(* CoDeSys 2.3.9.59 project: Proyecto_Maquina_Expendedora.pro *)
(* Libraries: Standard.LIB, Iecsfc.lib 2.6.14 11:37:46 *)

(* Global variable list: Global_Variables *)
VAR_GLOBAL
(*ENTRADAS*)
	boton1:BOOL;
	boton2:BOOL;
	boton3:BOOL;
	boton4:BOOL;
	boton5:BOOL;
	boton6:BOOL;
	diezcent:BOOL;
	cincucent:BOOL;
	ciencent:BOOL;
	selector1:BOOL;
	selector2:BOOL;
	selector3:BOOL;
	selector4:BOOL;
	selector5:BOOL;
	selector6:BOOL;
	M:BOOL;
	P:BOOL;
	devolucion:BOOL;
	atasca:BOOL;
	rearme:BOOL;
	auto:BOOL;
	recogeobjeto:BOOL;
	recogecambio:BOOL;
	seleccionado:INT;
	abrir:BOOL;
(*SALIDAS*)
	dispensador1:BOOL;
	dispensador2:BOOL;
	dispensador3:BOOL;
	dispensador4:BOOL;
	dispensador5:BOOL;
	dispensador6:BOOL;
	dinero:REAL;
	cambio:REAL;
	precio:REAL;
	display:REAL;
	puertacerrada: BOOL:=TRUE;
	objetoabajo: BOOL:=FALSE;
	fila1cae:BOOL;
	fila2cae:BOOL;
	fila3cae:BOOL;
	muestradinero:BOOL;
	muestracambio:BOOL;
	luzcae:BOOL;
	luzabajo:BOOL;
	resetobjeto:BOOL;
	emergencia:BOOL;
(*CONSTANTES*)
	precio1:REAL:=1.00;
	precio2:REAL:=1.30;
	precio3:REAL:=0.80;
	precio4:REAL:=1.60;
	precio5:REAL:=2.00;
	precio6:REAL:=0.90;

(*ESTADOS*)
	metedinero: BOOL;
	sacadinero: BOOL;
	caeobjeto: BOOL;
END_VAR

(* POU PLC_PRG, ST *)
PROGRAM PLC_PRG
VAR
	inicio:BOOL:=TRUE;
	camux: INT;
	camuy:INT;
	kinderx:INT;
	kindery:INT;
	chocox:INT;
	chocoy:INT;
	bullx:INT;
	bully:INT;
	mangox:INT;
	mangoy:INT;
	kitkatx:INT;
	kitkaty:INT;
	TEMPprecio: TON;
	apaga: F_TRIG;
	apagando: BOOL;
	color:DWORD;
END_VAR
(* Selector para mostrar dinero *)
IF (inicio) THEN
	precio:=0;
	inicio:=FALSE;
END_IF
apaga (CLK := (selector1 OR selector2 OR selector3 OR selector4 OR selector5 OR selector6));
IF apaga.Q THEN apagando := TRUE; END_IF
IF selector1 THEN precio := precio1; apagando := FALSE;
ELSIF selector2 THEN precio := precio2; apagando := FALSE;
ELSIF selector3 THEN precio := precio3; apagando := FALSE;
ELSIF selector4 THEN precio := precio4; apagando := FALSE;
ELSIF selector5 THEN precio := precio5; apagando := FALSE;
ELSIF selector6 THEN precio := precio6; apagando := FALSE;
END_IF

TEMPprecio(IN:= apagando, PT:=T#3s) ;
	IF TEMPprecio.Q THEN
		seleccionado := 0;
		precio := 0;
		apagando := FALSE;
	END_IF

(* Selector para mostrar dinero disponible o cambio dependiendo del estado *)
IF muestradinero THEN display := dinero;
ELSIF muestracambio THEN display := cambio;
ELSE display := 0.00;
END_IF

(* Dependiendo de cuál se elija, cae uno u otro *)
IF (auto AND NOT objetoabajo) OR NOT auto THEN
IF (dispensador1 = TRUE) AND (camuy<=545) THEN camuy := camuy + 10; fila1cae := TRUE;
	IF (camuy = 550) THEN
		objetoabajo:=TRUE;
		fila1cae:=FALSE;
	END_IF
ELSIF (dispensador2 = TRUE) AND (kindery <=545)THEN kindery := kindery + 10; fila1cae:=TRUE;
	IF (kindery = 550) THEN
		objetoabajo := TRUE;
		fila1cae:=FALSE;
	END_IF;
ELSIF (dispensador3 = TRUE) AND (chocoy<=395) THEN chocoy := chocoy + 10; fila2cae:=TRUE;
	IF (chocoy = 400) THEN
		objetoabajo:=TRUE;
		fila2cae:=FALSE;
	END_IF
ELSIF (dispensador4 = TRUE) AND (bully <= 395) THEN bully := bully + 10; fila2cae:=TRUE;
	IF (bully = 400) THEN
		objetoabajo:=TRUE;
		fila2cae:=FALSE;
	END_IF
ELSIF (dispensador5 = TRUE) AND (mangoy <= 255) THEN mangoy := mangoy + 10; fila3cae:=TRUE;
	IF (mangoy = 260) THEN
		objetoabajo:=TRUE;
		fila3cae:=FALSE;
	END_IF
ELSIF (dispensador6 = TRUE) AND (kitkaty <= 255) THEN kitkaty := kitkaty + 10; fila3cae:=TRUE;
	IF (kitkaty = 260) THEN
		objetoabajo:=TRUE;
		fila3cae:=FALSE;
	END_IF
ELSIF NOT (dispensador1 OR dispensador2 OR dispensador3 OR dispensador4 OR dispensador5 OR dispensador6) THEN
	fila1cae:=FALSE;
	fila2cae:=FALSE;
	fila3cae:=FALSE;
END_IF
END_IF
IF resetobjeto THEN
	camuy:=0;
	kindery:=0;
	chocoy:=0;
	bully:=0;
	mangoy:=0;
	kitkaty:=0;
	objetoabajo:=FALSE;
END_IF


(* Excepto cuando sale el cambio, si se selecciona un objeto y
 el dinero disponible es menor al necesario se muestra en rojo, 
 en caso contrario será en verde, usa BGR en vez de RGB *)
IF (muestradinero) THEN
	IF (apaga.Q) THEN color:=16#000000;
	ELSIF (ABS(dinero-precio) < 0.01) THEN color:=16#13D613;
	ELSE color:=16#1717D4;
	END_IF
ELSE color := 16#000000;
END_IF

PRG_Principal;
END_PROGRAM

(* POU PRG_Principal, ST *)
PROGRAM PRG_Principal
VAR
	camu:Modo_Auto;
	kinder:Modo_Auto;
	choco:Modo_Auto;
	bull:Modo_Auto;
	mango:Modo_Auto;
	kitkat:Modo_Auto;
END_VAR
Calcula_Dinero;
IF atasca OR emergencia THEN
	camu(selector:=selector1,SFCRESET:=TRUE,dispensador=>dispensador1);
	kinder(selector:=selector2,SFCRESET:=TRUE,dispensador=>dispensador2);
	choco(selector:=selector3,SFCRESET:=TRUE,dispensador=>dispensador3);
	bull(selector:=selector4,SFCRESET:=TRUE,dispensador=>dispensador4);
	mango(selector:=selector5,SFCRESET:=TRUE,dispensador=>dispensador5);
	kitkat(selector:=selector6,SFCRESET:=TRUE,dispensador=>dispensador6);
	Modo_Emergencia(SFCRESET:=FALSE);
ELSE
	Modo_Emergencia(SFCRESET:=TRUE);
	IF auto THEN
			camu(selector:=selector1,SFCRESET:=FALSE,dispensador=>dispensador1);
			kinder(selector:=selector2,SFCRESET:=FALSE,dispensador=>dispensador2);
			choco(selector:=selector3,SFCRESET:=FALSE,dispensador=>dispensador3);
			bull(selector:=selector4,SFCRESET:=FALSE,dispensador=>dispensador4);
			mango(selector:=selector5,SFCRESET:=FALSE,dispensador=>dispensador5);
			kitkat(selector:=selector6,SFCRESET:=FALSE,dispensador=>dispensador6);
	ELSE
			camu(selector:=selector1,SFCRESET:=TRUE,dispensador=>dispensador1);
			kinder(selector:=selector2,SFCRESET:=TRUE,dispensador=>dispensador2);
			choco(selector:=selector3,SFCRESET:=TRUE,dispensador=>dispensador3);
			bull(selector:=selector4,SFCRESET:=TRUE,dispensador=>dispensador4);
			mango(selector:=selector5,SFCRESET:=TRUE,dispensador=>dispensador5);
			kitkat(selector:=selector6,SFCRESET:=TRUE,dispensador=>dispensador6);
			Modo_Manual;
	END_IF
END_IF
END_PROGRAM

(* POU Modo_Auto, SFC *)
FUNCTION_BLOCK Modo_Auto
VAR_INPUT
	selector:BOOL;
	SFCRESET:BOOL;
END_VAR
VAR_OUTPUT
	dispensador:BOOL;
END_VAR
VAR
	marcha: BOOL;
	puerta:BOOL;
END_VAR
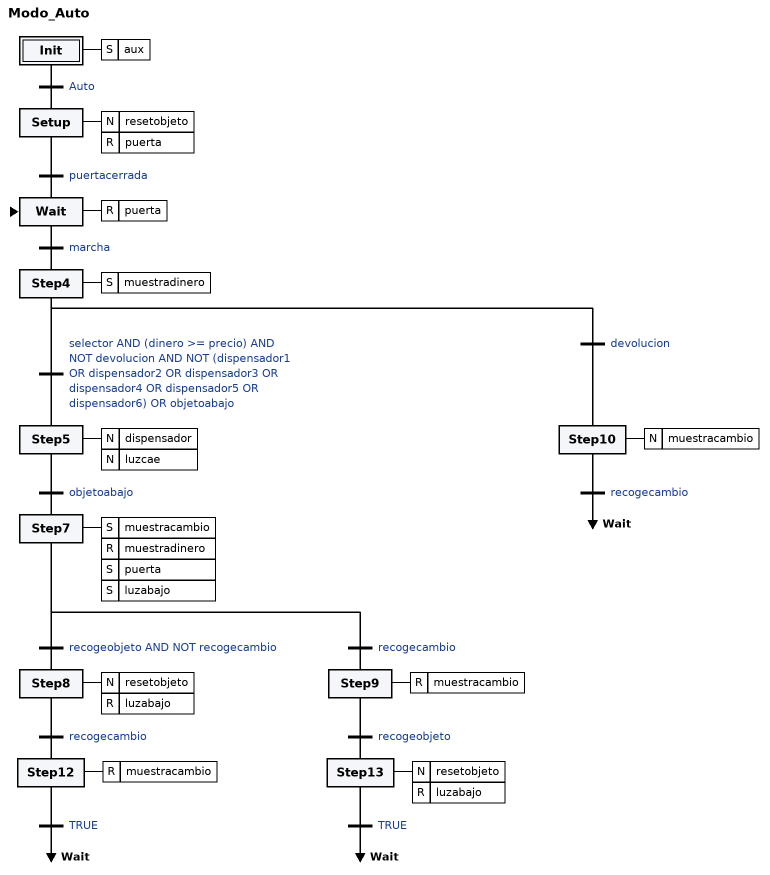
INITIAL_STEP Init:
	aux(S);
END_STEP
TRANSITION FROM Init TO Setup := Auto;
END_TRANSITION
STEP Setup:
	resetobjeto(N);
	puerta(R);
END_STEP
TRANSITION FROM Setup TO Wait := puertacerrada;
END_TRANSITION
STEP Wait:
	puerta(R);
END_STEP
TRANSITION FROM Wait TO Step4 := marcha;
END_TRANSITION
STEP Step4:
	muestradinero(S);
END_STEP
TRANSITION FROM Step4 TO Step5 := selector AND (dinero >= precio) AND NOT devolucion AND NOT (dispensador1 OR dispensador2 OR dispensador3 OR dispensador4 OR dispensador5 OR dispensador6) OR objetoabajo;
END_TRANSITION
TRANSITION FROM Step4 TO Step10 := devolucion;
END_TRANSITION
STEP Step10:
	muestracambio(N);
END_STEP
TRANSITION FROM Step10 TO Wait := recogecambio;
END_TRANSITION
STEP Step5:
	dispensador(N);
	luzcae(N);
END_STEP
TRANSITION FROM Step5 TO Step7 := objetoabajo;
END_TRANSITION
STEP Step7:
	muestracambio(S);
	muestradinero(R);
	puerta(S);
	luzabajo(S);
END_STEP
TRANSITION FROM Step7 TO Step8 := recogeobjeto AND NOT recogecambio;
END_TRANSITION
TRANSITION FROM Step7 TO Step9 := recogecambio;
END_TRANSITION
STEP Step8:
	resetobjeto(N);
	luzabajo(R);
END_STEP
TRANSITION FROM Step8 TO Step12 := recogecambio;
END_TRANSITION
STEP Step12:
	muestracambio(R);
END_STEP
TRANSITION FROM Step12 TO Wait := TRUE;
END_TRANSITION
STEP Step9:
	muestracambio(R);
END_STEP
TRANSITION FROM Step9 TO Step13 := recogeobjeto;
END_TRANSITION
STEP Step13:
	resetobjeto(N);
	luzabajo(R);
END_STEP
TRANSITION FROM Step13 TO Wait := TRUE;
END_TRANSITION
END_FUNCTION_BLOCK
ACTION aux:
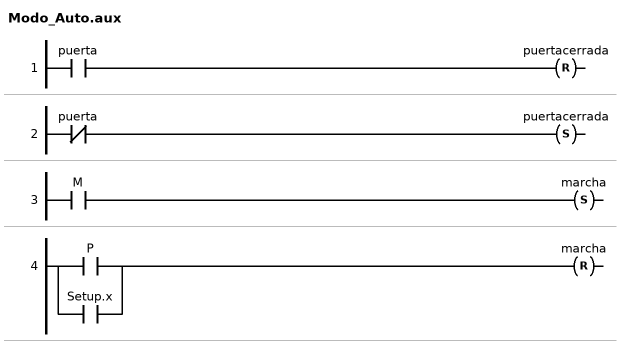
_LD_ (* Ladder Diagram *)
NETWORK 1
	[puerta] --- (R puertacerrada)
NETWORK 2
	[/puerta] --- (S puertacerrada)
NETWORK 3
	[M] --- (S marcha)
NETWORK 4
	{ [P] | [Setup.x] } --- (R marcha)
_END_LD_
(* the same logic as Structured Text *)
(* Network 1 *)
IF puerta THEN puertacerrada := FALSE; END_IF;
(* Network 2 *)
IF NOT puerta THEN puertacerrada := TRUE; END_IF;
(* Network 3 *)
IF M THEN marcha := TRUE; END_IF;
(* Network 4 *)
IF P OR Setup.x THEN marcha := FALSE; END_IF;
END_ACTION

(* POU Calcula_Dinero, ST *)
PROGRAM Calcula_Dinero
VAR
	precioact:REAL;
	diez:F_TRIG;
	cincuenta:F_TRIG;
	cien:F_TRIG;
END_VAR
diez(clk:=diezcent);
cincuenta(clk:=cincucent);
cien(clk:=ciencent);
IF muestradinero AND auto THEN
	cambio:=0;
	IF diez.Q THEN
		dinero:=dinero+0.10;
	ELSIF cincuenta.Q THEN
		dinero:=dinero+0.5;
	ELSIF cien.Q THEN
		dinero:=dinero+1;
	END_IF
	IF precioact <=0.01 THEN
		IF dispensador1 THEN
			precioact:=precio1;
		ELSIF dispensador2 THEN
			precioact:=precio2;
		ELSIF dispensador3 THEN
			precioact:=precio3;
		ELSIF dispensador4 THEN
			precioact:=precio4;
		ELSIF dispensador5 THEN
			precioact:=precio5;
		ELSIF dispensador6 THEN
			precioact:=precio6;
		END_IF
	END_IF
ELSIF muestracambio AND auto THEN
	IF precioact >= 0.1 AND cambio <= 0.01 AND precioact <= 67 THEN
		cambio:=dinero-precioact;
		precioact:=69;
	ELSIF precioact <= 0.01 AND cambio<= 0.01THEN
		cambio:=dinero;
	END_IF
ELSE
	dinero:=0;
	cambio:=0;
	precioact:=0;
END_IF
END_PROGRAM

(* POU Modo_Emergencia, SFC *)
PROGRAM Modo_Emergencia
VAR_INPUT
	SFCRESET:BOOL;
END_VAR
VAR
END_VAR
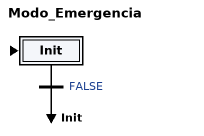
INITIAL_STEP Init:
END_STEP
TRANSITION FROM Init TO Init := FALSE;
END_TRANSITION
END_PROGRAM

(* POU Modo_Manual, LD *)
PROGRAM Modo_Manual
VAR
END_VAR
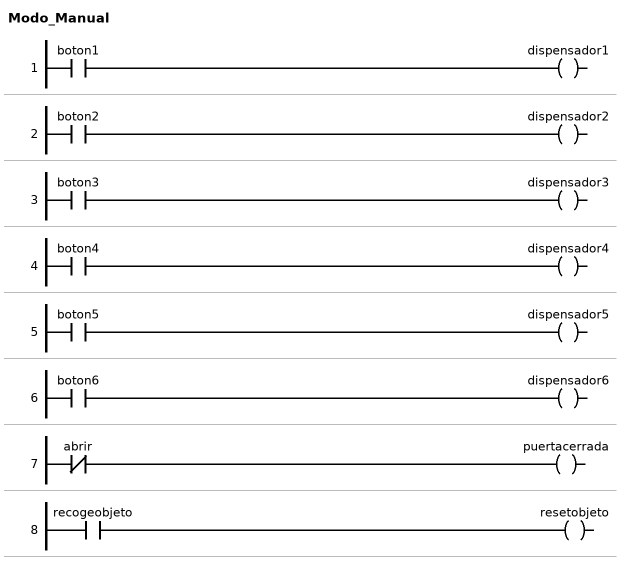
_LD_ (* Ladder Diagram *)
NETWORK 1
	[boton1] --- (dispensador1)
NETWORK 2
	[boton2] --- (dispensador2)
NETWORK 3
	[boton3] --- (dispensador3)
NETWORK 4
	[boton4] --- (dispensador4)
NETWORK 5
	[boton5] --- (dispensador5)
NETWORK 6
	[boton6] --- (dispensador6)
NETWORK 7
	[/abrir] --- (puertacerrada)
NETWORK 8
	[recogeobjeto] --- (resetobjeto)
_END_LD_
(* the same logic as Structured Text *)
(* Network 1 *)
dispensador1 := boton1;
(* Network 2 *)
dispensador2 := boton2;
(* Network 3 *)
dispensador3 := boton3;
(* Network 4 *)
dispensador4 := boton4;
(* Network 5 *)
dispensador5 := boton5;
(* Network 6 *)
dispensador6 := boton6;
(* Network 7 *)
puertacerrada := NOT abrir;
(* Network 8 *)
resetobjeto := recogeobjeto;
END_PROGRAM

(* Visualisation Maquina
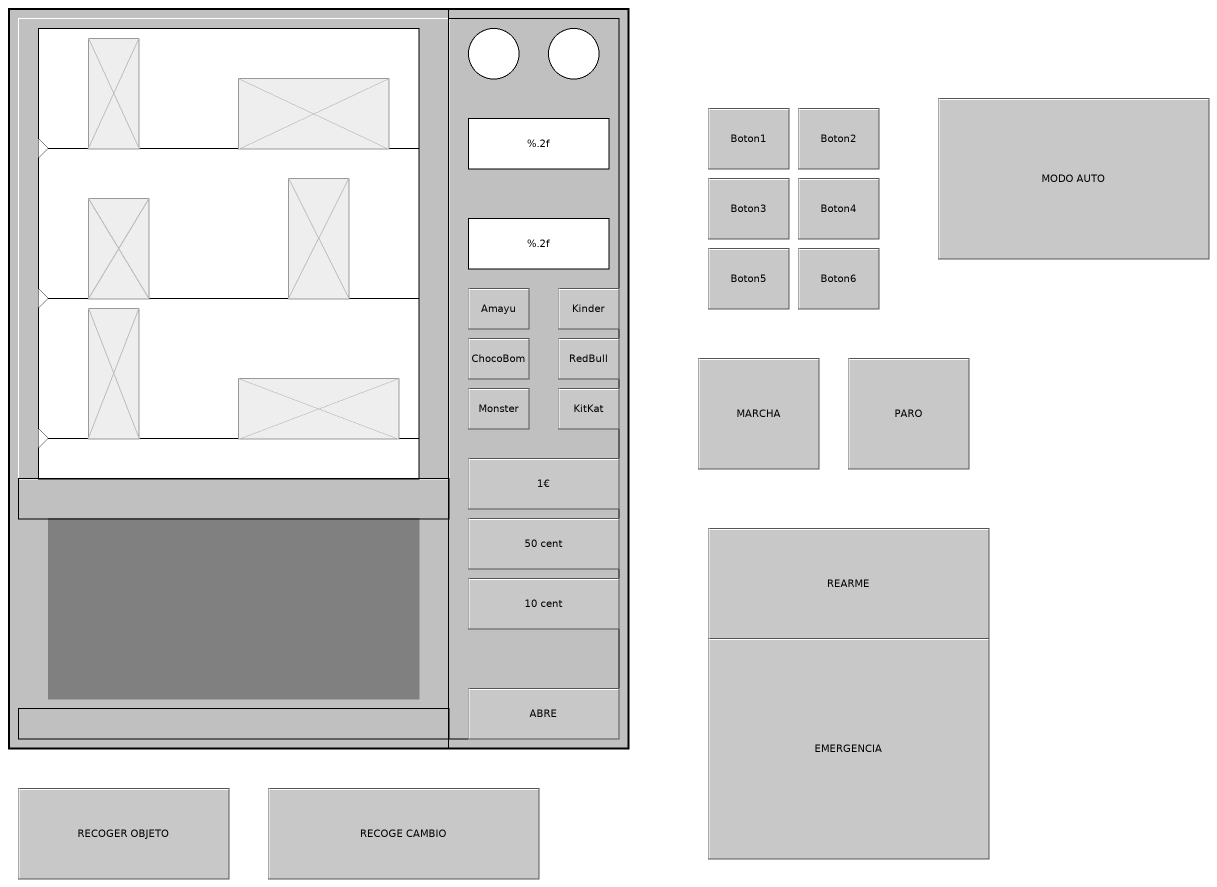
button at (480,290)-(541,331): text "Amayu"; taps .selector1
button at (570,290)-(631,331): text "Kinder"; taps .selector2
button at (570,390)-(631,431): text "KitKat"; taps .selector6
button at (480,390)-(541,431): text "Monster"; taps .selector5
button at (570,340)-(631,381): text "RedBull"; taps .selector4
button at (480,340)-(541,381): text "ChocoBom"; taps .selector3
rectangle at (480,120)-(621,171): text "%.2f"; shows .precio
rectangle at (480,220)-(621,271): text "%.2f"; shows .display
bitmap at (100,310)-(151,441): images\mango.jpg
bitmap at (100,200)-(161,301): images\chocobom.jpg
bitmap at (100,40)-(151,151): images\amayu.jpg
bitmap at (250,380)-(411,441): images\kitkat.jpg
bitmap at (300,180)-(361,301): images\redredbull.jpg
bitmap at (250,80)-(401,151): images\kinderbueno.jpg
rectangle at (60,520)-(431,701): alarm colour if .puertacerrada
button at (480,690)-(631,741): text "ABRE"; toggles abrir
ellipse at (480,30)-(531,81): alarm colour if luzcae
ellipse at (560,30)-(611,81): alarm colour if luzabajo
polygon at (50,140)-(60,160): alarm colour if fila1cae
polygon at (50,290)-(60,310): alarm colour if fila2cae
polygon at (50,430)-(60,450): alarm colour if fila3cae
button at (480,460)-(631,511): text "1€"; taps ciencent
button at (480,520)-(631,571): text "50 cent"; taps cincucent
button at (480,580)-(631,631): text "10 cent"; taps diezcent
button at (720,110)-(801,171): text "Boton1"; taps Boton1
button at (720,180)-(801,241): text "Boton3"; taps Boton3
button at (810,110)-(891,171): text "Boton2"; taps Boton2
button at (810,180)-(891,241): text "Boton4"; taps Boton4
button at (720,250)-(801,311): text "Boton5"; taps Boton5
button at (810,250)-(891,311): text "Boton6"; taps Boton6
button at (710,360)-(831,471): text "MARCHA"; taps M
button at (860,360)-(981,471): text "PARO"; taps P
button at (720,530)-(1001,641): text "REARME"; taps rearme
button at (720,640)-(1001,861): text "EMERGENCIA"; toggles atasca
button at (950,100)-(1221,261): text "MODO AUTO"; toggles auto
button at (30,790)-(241,881): text "RECOGER OBJETO"; taps recogeobjeto
button at (280,790)-(551,881): text "RECOGE CAMBIO"; taps recogecambio
11 more shapes without text or variables
*)
